    User Values are:
    0 = Not Used, 1 = FIC-21-1, 2 = EV-2, 3 = EV-3, 4 = AG-4, 5 = FIC-21-2, 6 = FIC-21-3, 7 = FIC-21-4, 8 = FIC-46-1, 9 = EV-42, 10 = EV-20
  N24:12: This Rung Calculates
    the Range Values for PID Statements, Analog Inputs and Analog Outputs
    These are used Elsewhere in PLC Logic to calulate either
    other Units
    (PID Statement Inputs, Analog Output Values, etc)
  N24:20: This Rung Calculates the PLC Ranges as Shown
    For use elsewhere in the PLC Program
  N50:0/0: This Rung Stops EV-1 Rotor Drive
    when the operator presses the EV-1 PB
    AND the motor is Off
    OR
    The Interlocks are NOT satisfied
  N50:2/0: This Rung determines the status of the Interlocks for EV-1 Rotor Drive
  N50:4/0: This rung sets a 1-shot bit whenever EV-1 Rotor Drive
    is Started
  N50:5/13: This rung sets a 1-shot bit whenever EH-24 Hot Oil Heater
    HMI Start/Stop PB
    is Pressed
  N50:6/0: This rung sets a 1-shot bit whenever EV-1 Rotor Drive
    is Stopped
  N50:15/11: This Rung Resets All
    HMI PB's to
    0 State to allow their next use to be detected
    (This is required due to iFIX's inability to generate momentary PB's, not required for PanelView Plus)
  N50:16/11: This Rung Generates a 1-shot
    whenever the Operator
    presses the FIC-21-1 Output Select PB
  N50:20: This rung resets any
    iFIX Momentary PB's to 0
    (ifix does not have momentary PB Feature)
  N50:41/14: This rung sets a 1-shot bit whenever
    the EV-2 Residue
    Calculate Flow Rate PB
    is Pressed
  N61:0/[N23:82]: This Rung Starts EV-2 Rotor Drive
    when the operator presses the EV-2 PB
    AND
    the Interlocks are satisfied and the motor is Off
  N101:20/0: DELETE THIS RUN FOR REAL PLC
  N213:1: This Rung Converts the Output from
    PIC-28-1
    Steam Pressure Controller
    to Open PV-28-1 (Steam Valve) Between 0% to 100% .
    PV-28-1 Fails Closed
  N213:3: This Rung Split Ranges the Output from
    TIC-11-1
    Tempered Water Loop No-1
    to Close TV-11-1 (Cooling Valve) Between 0% to 50% while keeping TV-11-2 (Heating Valve) Closed.
    then
    to Open TV-11-2 (Heating Valve) Between 50% to 100% while keeping TV-11-1 (Cooling valve) Closed.
    At  50%, Both Valves are Closed
      TV-11-1 Fails Open, TV-11-2 Fails Closed
  N214:0: This Rung Converts the Output from
    TIC-12-1
    Tempered Water Loop No-2
    to Close TV-12-1 (Cooling Valve) Between 0% to 100% .
    TV-12-1 Fails Open
  N214:1: This Rung Converts the Output from
    TIC-15-1
    Tempered Oil Loop No-1
    to Open TV-15-1 (Heating Valve) Between 0% to 100% .
    TV-15-1 Fails Closed
  N214:3: This Rung Converts the Output from
    TIC-24-1
    Hot Oil Loop
    to Increase the Firing Rate of TY-24-1 (Heater SCR Controller) Between 0% to 100% .
    TY-24-1 is Off 100% at 0%, On 50% of time at 50% and On 100% of time at 100%.
  N215:0: This Rung Sends the
    EV-2 Rotor Speed Setpoint
    to the VFD which controls its speed.
    A 1-shot is used when the motor is started to set an initial speed
    A 1-shot is also used when it is stopped to reset the speed to 0.0
    and the last rung actually passed the speed signal to the analog output module which sontrols the motors speed
  N215:1: This Rung Sends the
    EV-3 Rotor Speed Setpoint
    to the VFD which controls its speed.
    A 1-shot is used when the motor is started to set an initial speed
    A 1-shot is also used when it is stopped to reset the speed to 0.0
    and the last rung actually passed the speed signal to the analog output module which sontrols the motors speed
  N215:2: This Rung Sends the
    AG-4 Agitator Speed Setpoint
    to the VFD which controls its speed.
    A 1-shot is used when the motor is started to set an initial speed
    A 1-shot is also used when it is stopped to reset the speed to 0.0
    and the last rung actually passed the speed signal to the analog output module which sontrols the motors speed
  N216:1: This Rung Moves the
    FIC-21-1 PID Output to the
    Selected Pump VFD Speed Control Based on which Pump is Connected to the Feed Flow Loop
  N216:3: This Rung Moves the
    PIC-30-1 PID Output to Pump PU-30's VFD Speed Control
  N218:0: This Rung Copies Setup Data for all TE's
    to their Output Addresses when the PLC is first placed in the Run Mode
    This Information determines that the TE data returned from the Input modules will
    use °C Units for a Type "J" Thermocouple
  O:6.16/0: This Rung Starts PU-13 Tempered Oil Pump No-2
    when the operator presses the PU-13 PB
    AND
    the Interlocks are satisfied and the motor is Off
  O:6.19/4: This Rung Starts PU-13 Tempered Oil Pump No-2
    when the operator presses the PU-13 PB
    AND
    the Interlocks are satisfied and the motor is Off
  O:15.0: This Rung Controls the Status and Speed of
    VFD02
    if it's controls are enabled
  O:15.1: This Rung Controls the Status and Speed of
    VFD03
    if it's controls are enabled
  O:15.2: This Rung Controls the Status and Speed of
    VFD04
    if it's controls are enabled
  O:15.3: This Rung Controls the Status and Speed of
    VFD01
    if it's controls are enabled
  O:23.0/0: This Rung Stops EV-1 Rotor Drive
    when the operator presses the EV-1 PB
    AND the motor is Off
    OR
    The Interlocks are NOT satisfied
  O:23.0/11: This Rung Starts PU-23 Hot Oil Pump
    when the operator presses the PU-23 PB
    AND
    the Interlocks are satisfied and the motor is Off
  O:23.0/12: This Rung Starts EH-24 Hot Oil Heater
    when the operator presses the EH-24 PB
    AND the Heater is Off
    AND
    The Interlocks are satisfied
  Q62:1: This Rung Enables EH-24, Hot Oil Heater
    when the operator presses the EH-24 PB
    AND
    the Interlocks are satisfied and the Contatcer is Off
     (The Jump Stattement is required since this device does Not have a feedback connection from contactor to indicate actual status,
    because of this, an internal bit is used.  When an internal bit is used, the next statement (Stop/disable)
    will immediantely be executed, resulting in the motor/contactor not being de-energized.  The Jump statement eliminates this problem)
  Q64:1: This Rung Enables EH-27, Hot Oil SuperHeater
    when the operator presses the EH-27 PB
    AND
    the Interlocks are satisfied and EH-27 is disabled
      (The Jump Stattement is required since this device does Not have a feedback connection from contactor to indicate actual status,
    because of this, an internal bit is used.  When an internal bit is used, the next statement (Stop/disable)
    will immediantely be executed, resulting in the motor/contactor not being de-energized.  The Jump statement eliminates this problem)
  T4:31: This Rung Sets a bit when
    PT-26-1 is less than PSL-26-1's Setpoint.
    Used to enable VB-26
  T51:0: This run starts a timer whenever EV-1 Rotor Drive
    is started to verify that it actually starts within 5 sec's
    If Not, then it is assumed that the motor's O.l.s have tripped
  T51:1: This run starts a timer whenever EV-2 Rotor Drive
    is started to verify that it actually starts within 5 sec's
    If Not, then it is assumed that the motor's O.l.s have tripped
  T51:2: This run starts a timer whenever EV-3 Rotor Drive
    is started to verify that it actually starts within 5 sec's
    If Not, then it is assumed that the motor's O.l.s have tripped
  T51:3: This run starts a timer whenever AG-4 Feed Tank Agitator
    is started to verify that it actually starts within 5 sec's
    If Not, then it is assumed that the motor's O.l.s have tripped
  T51:4: This run starts a timer whenever VP-9 Beach-Ross Vacuum Pump
    is started to verify that it actually starts within 5 sec's
    If Not, then it is assumed that the motor's O.l.s have tripped
  T51:5: This run starts a timer whenever VP-10 Kinney Vacuum Pump
    is started to verify that it actually starts within 5 sec's
    If Not, then it is assumed that the motor's O.l.s have tripped
  T51:6: This run starts a timer whenever PU-11 Tempered Water Pump No-1
    is started to verify that it actually starts within 5 sec's
    If Not, then it is assumed that the motor's O.l.s have tripped
  T51:7: This run starts a timer whenever PU-12 Tempered Water Pump No-2
    is started to verify that it actually starts within 5 sec's
    If Not, then it is assumed that the motor's O.l.s have tripped
  T51:8: This run starts a timer whenever PU-15 Tempered Oil Pump
    is started to verify that it actually starts within 5 sec's
    If Not, then it is assumed that the motor's O.l.s have tripped
  T51:9: This run starts a timer whenever PU-21 Feed Pump No-1
    is started to verify that it actually starts within 5 sec's
    If Not, then it is assumed that the motor's O.l.s have tripped
  T51:10: This run starts a timer whenever PU-22 Feed Pump No-2
    is started to verify that it actually starts within 5 sec's
    If Not, then it is assumed that the motor's O.l.s have tripped
  T51:11: This run starts a timer whenever PU-23 Hot Oil Pump
    is started to verify that it actually starts within 5 sec's
    If Not, then it is assumed that the motor's O.l.s have tripped
  T51:13: This run starts a timer whenever VB-26 Roots Vacuum Blower
    is started to verify that it actually starts within 5 sec's
    If Not, then it is assumed that the motor's O.l.s have tripped
  T51:15: This run starts a timer whenever PU-30 City Water Booster Pump
    is started to verify that it actually starts within 5 sec's
    If Not, then it is assumed that the motor's O.l.s have tripped
  T51:16: This run starts a timer whenever  VB-35 TutHill Vacuum Blower
    is started to verify that it actually starts within 5 sec's
    If Not, then it is assumed that the motor's O.l.s have tripped
  U:3: This Rung Calls the Subroutine Files Listed
  U:10: This Rung Calls the Subroutine Files Listed
  U:31: This Rung Calls the Subroutine Files Listed
  U:59: This Rung Calls the Subroutine Files Listed
  U:66: This Rung Calls the Subroutine Files Listed
  U:101: DELETE THIS RUNG AND FILE WHEN USING THE REAL PLC CONFIGURATION WITH REAL I/O

REVISION NOTES
  0: Totalizer Updates for Harting Test

DATA TABLE (non-zero values as saved)
DATA B3
% B3:0 % 0X007E 0X0000 0X0000 0X0000 0X0000 0X000C 0X0000 0X0000 0X0000 0X0000
% B3:10 % 0X9000 0X0000 0X0002 0X0000 0X0000 0X0000 0X0000 0X0000 0X0000 0X0000
% B3:20 % 0X0000 0X0000 0X0002 0X0000 0X0000 0X0000 0X0000 0X0000 0X0000 0X0000
% B3:30 % 0X0009 0X0000 0X0000 0X0000 0X0009 0X0000 0X0000 0X0000 0X0000 0X0000
% B3:70 % 0X0028 0X0000 0X0000 0X0000 0X0000 0X0000 0X0000 0X0000 0X0000 0X0000
DATA T4
% .PRE .ACC %
% T4:0 % 150 0
% T4:1 % 3000 1418
% T4:2 % 3600 1529
% T4:3 % 1000 0
% T4:4 % 100 0
% T4:6 % 1 0
% T4:11 % 6000 0
% T4:12 % 6000 0
% T4:13 % 6000 0
% T4:14 % 6000 0
% T4:21 % 10 10
% T4:22 % 50 30
% T4:23 % 10 10
% T4:24 % 50 30
% T4:25 % 30 30
% T4:26 % 12 6
% T4:30 % 5 0
% T4:31 % 5 5
% T4:32 % 2 0
% T4:34 % 5 0
% T4:35 % 1 0
DATA C5
% .PRE .ACC %
% C5:0 % 3600 1446
% C5:1 % 16000 -19876
% C5:2 % 16000 0
% C5:3 % 16000 21413
% C5:4 % 16000 21419
% C5:5 % 16000 21249
% C5:6 % 16000 21298
% C5:7 % 16000 2
% C5:8 % 16000 22936
% C5:11 % 600 0
% C5:12 % 600 0
% C5:13 % 600 600
% C5:14 % 600 0
DATA N7
% N7:0 % 4 7 2014 0 0 0 0 0 0 0
DATA F8
% F8:0 % 100 200 0 0 0
DATA N11
% N11:0 % 0 277 253 259 300 7599 7599 7599 7599 7599
% N11:10 % 267 274 275 298 282 7599 7599 7599 7599 315
% N11:20 % 315 263 264 265 256 275 7599 264 265 170
% N11:30 % 187 204 259 286 283 282 284 0 0 0
% N11:100 % 6 15152 0 16383 16383 12197 0 0 0 16383
% N11:120 % 1500 50 1950 600 50 10000 750 0 10000 10000
% N11:130 % 0 13313 8018 1564 0 0 0 0 0 0
% N11:150 % 0 2000 1000 1500 0 0 0 0 0 0
% N11:190 % 0 1000 0 0 0 0 0 0 0 0
% N11:220 % 0 5000 6000 5000 6000 6000 6000 0 0 0
DATA N12
% N12:0 % 0 170 187 204 259 286 283 282 284 0
% N12:10 % 128 0 0 0 0 0 0 0 0 0
% N12:20 % 0 0 8 8 8 8 8 8 0 0
% N12:100 % 0 0 0 0 0 0 0 0 -32768 0
% N12:110 % 0 0 0 0 0 0 0 0 -32768 0
% N12:120 % 15 0 0 0 0 0 0 0 0 0
DATA N13
% N13:0 % 0 3136 3136 3136 3136 3136 3136 3136 3136 3136
% N13:10 % 3136 3136 3136 3136 3136 3136 3136 3136 3136 3136
% N13:20 % 3136 3136 3136 3136 3136 3136 3136 3136 3136 0
% N13:30 % 0 13107 13107 0 0 0 0 0 0 0
% N13:40 % 255 0 0 0 0 0 0 0 0 0
% N13:50 % 0 0 0 0 15 3840 0 0 0 0
% N13:70 % 0 0 0 0 15 3840 0 0 0 0
% N13:100 % -256 0 0 0 0 0 0 0 0 0
% N13:110 % -256 0 0 0 0 0 0 0 0 0
% N13:120 % 0 0 0 0 15 3840 0 0 0 0
DATA F14
% F14:5 % 40 30 0 0 0
% F14:10 % 45 0 0 0 0
DATA N15
% N15:0 % -24566 0 0 8 5 10 0 6000 0 0
% N15:10 % 0 60 0 15 0 0 0 0 -5805 0
% N15:20 % 0 0 0 0 0 40 1 0 5000 7500
% N15:30 % -24574 0 0 7 5 11 0 6000 0 0
% N15:40 % 0 60 0 15 0 0 0 0 7241 0
% N15:60 % -24570 0 0 50 3 0 0 1950 0 0
% N15:70 % 0 100 0 15 0 0 100 16383 0 0
% N15:80 % 0 0 0 0 0 0 0 2500 5000 7500
% N15:90 % -24570 0 7444 100 10 0 0 10000 0 0
% N15:100 % 0 100 0 15 7444 0 80 13086 29382 2
% N15:110 % -1456 0 7444 0 12197 0 0 0 0 0
% N15:150 % -24318 0 1580 2 5 0 0 2000 0 10
% N15:160 % 0 100 0 15 1580 2 50 8192 -12210 3
% N15:170 % 10592 0 1582 0 13313 0 0 500 1000 1500
% N15:180 % -24566 0 377 20 10 0 0 1000 0 0
% N15:190 % 0 83 0 15 377 5 0 -156 -28170 1
% N15:200 % -31472 0 381 0 8018 0 0 250 500 750
DATA N16
% N16:0 % -24566 0 0 8 5 10 0 6000 0 0
% N16:10 % 0 60 0 15 0 0 0 0 -24274 0
% N16:20 % 0 0 0 0 0 0 0 950 1900 2850
% N16:30 % -24314 0 0 10 5 0 0 5000 0 0
% N16:40 % 0 60 0 15 0 0 0 0 -2178 0
% N16:50 % 0 0 0 0 0 0 0 1500 3000 4500
% N16:60 % -24318 0 143 100 5 0 0 1500 0 0
% N16:70 % 0 60 0 15 143 0 0 0 9388 0
% N16:80 % 25024 0 143 0 1564 0 0 750 1500 2250
% N16:150 % -24570 0 0 100 3 0 0 1000 0 0
% N16:160 % 0 60 0 15 0 0 0 0 0 0
DATA N17
% N17:0 % -24318 0 170 15 3 0 11468 2000 0 0
% N17:10 % 0 100 0 15 170 0 50 -3276 30726 0
% N17:20 % 22288 0 170 0 1393 50 0 0 0 0
% N17:30 % -24318 0 259 20 3 0 0 2000 0 0
% N17:40 % 0 100 0 15 259 0 50 8192 25776 0
% N17:50 % -31584 0 259 0 2122 50 0 0 0 0
% N17:60 % -24318 0 286 250 20 5 0 3500 0 0
% N17:70 % 0 100 0 15 286 0 0 40 20578 0
% N17:80 % 21485 0 286 0 1325 0 0 0 0 0
% N17:90 % -24566 0 283 900 400 0 0 3500 0 0
% N17:100 % 0 100 0 15 283 0 0 450 -2237 0
% N17:110 % 21264 0 283 0 1329 0 3430 0 0 0
% N17:120 % -24574 0 280 30 30 0 0 3500 0 0
% N17:130 % 0 100 0 15 280 0 0 3 1632 0
% N17:140 % 20976 0 280 0 1320 0 0 0 0 0
% N17:150 % -24318 0 264 100 30 5 0 3500 0 0
% N17:160 % 0 100 0 15 264 0 0 0 -10202 0
% N17:170 % 19776 0 264 0 1236 0 0 0 0 0
DATA N18
% N18:0 % 0 0 0 0 0 16383 13106 0 8192 0
% N18:10 % 0 0 16383 16383 0 0 0 0 0 0
% N18:20 % 0 8192 8192 0 0 0 0 0 0 0
DATA N20
% N20:0 % 0 51 51 0 0 0 0 0 0 0
% N20:30 % -5 -5 -5 -5 -5 -5 -5 -5 0 0
DATA F21
% F21:0 % 0 27.7 25.3 25.9 30
% F21:5 % 759.9 759.9 759.9 759.9 759.9
% F21:10 % 26.7 27.4 27.5 29.8 28.2
% F21:15 % 759.9 759.9 759.9 759.9 31.5
% F21:20 % 31.5 26.3 26.4 26.5 25.6
% F21:25 % 27.5 759.9 26.4 26.5 17
% F21:30 % 18.7 20.4 25.9 28.6 28.3
% F21:35 % 28.2 28.4 0 0 0
% F21:50 % 0 162.521 48.93941 14.31787 0
% F21:60 % 0 -0.1526019 5.859911 -0.2289028 0
% F21:65 % 0 0 0.01526019 -50.02289 -15.00229
% F21:70 % 0.3815047 4.624218 -48.74256 61.95483 5.156798
% F21:75 % 744.4682 77.43781 0 -0.3571429 1258.202
% F21:80 % -250.0381 3604.48 2621.44 0.025 0
% F21:95 % 0 0 83417.15 0.0038 205.7111
% F21:120 % 0 0.01159703 0.01373333 -0.0006103702 0.002746666
% F21:125 % 0 0.003204639 0 0 0.001495453
% F21:130 % 0 -0.07630093 -0.04578056 -0.1144514 -9.385015
% F21:135 % 0 -2.563711 0 0 0
% F21:140 % 0 0.2499619 0.4996948 0.4938959 0.4841294
% F21:145 % 0.4997711 0.4937433 0 0 0
% F21:160 % 29.75736 0 0 0 0
% F21:170 % 0 0 0 0.002929777 0.003906369
% F21:175 % 0 0 0 0.001953185 0
% F21:180 % 0.007202368 0 0 0 0
% F21:195 % 0 0 0 0 199.76
% F21:200 % 0 -25.00381 0 0 0
% F21:205 % 0 -50.00763 0 0 0
DATA F22
% F22:0 % 22.22 27.45 0 0 0
% F22:10 % 0 4.624218 0.3815047 61.95483 0
% F22:20 % 0 0.3815047 0.3815047 0.3815047 0
% F22:50 % 0 26.7 26.4 26.5 26.3
% F22:55 % 0 26.7 27.5 27.7 0
% F22:60 % 0 28.2 759.9 759.9 27.4
% F22:65 % 26.7 25.6 31.5 26.5 0
% F22:70 % 0 26.3 26.7 26.5 25.6
% F22:75 % 27.5 759.9 26.4 26.5 0
% F22:90 % 0 26.7 25.9 28.6 28.3
% F22:95 % 28.2 28.4 0 0 0
% F22:100 % 0 759.9 759.9 25.9 27.5
% F22:110 % 0 25.3 27.7 0 0
% F22:120 % 0 17 0 0 0
% F22:130 % 0 25.9 0 0 0
% F22:140 % 0 28.3 28.2 26.4 0
% F22:180 % 0 28.4 0 0 0
% F22:190 % 0 759.9 31.5 0 0
% F22:200 % 26.4 26.4 26.4 26.4 27.5
% F22:205 % 0 27.5 31.5 0 0
% F22:210 % 0 -0.04578056 -0.07630093 0 0
% F22:220 % 0 -0.1144514 0 -0.07630093 0
% F22:230 % 0 -0.1144514 -0.1144514 -0.1144514 0
DATA N23
% N23:0 % 0 24 6 10 36 1 0 0 0 0
% N23:10 % 0 2 5 0 0 0 0 0 0 0
% N23:20 % 0 2 5 6 3 0 0 0 0 0
% N23:30 % 0 2 1 0 3 0 1 3 3 3
% N23:40 % 7 132 131 130 133 130 131 133 133 133
% N23:50 % 0 1 0 3 0 0 0 0 0 0
% N23:60 % 11 71 70 73 70 70 70 0 0 0
% N23:70 % 8 0 0 1 0 8 0 0 0 0
% N23:80 % 9 0 2 3 4 0 5 0 0 0
% N23:90 % 0 6 2 3 4 10 0 0 8 0
% N23:100 % 0 10 27 23 21 0 10 25 1 14
% N23:110 % 15 16 11 10 24 19 23 21 10 23
% N23:120 % 24 25 26 27 28 0 0 0 10 32
% N23:130 % 33 34 5 6 3 25 2 1 0 0
% N23:140 % 29 3 34 0 0 0 0 0 0 0
% N23:150 % 0 0 36 17 20 0 0 35 36 0
% N23:160 % 12 19 0 0 0 0 0 0 0 0
% N23:170 % 35 27 27 27 27 27 25 0 0 0
% N23:210 % 0 130 130 130 130 130 130 0 0 0
% N23:220 % 2 1 0 0 0 0 0 0 0 0
% N23:240 % 0 1 1 1 1 0 0 0 0 0
% N23:250 % 0 4 0 0 0 0
DATA N24
% N24:0 % 3277 16383 13106 0 0 0 32767 32767 0 0
% N24:10 % 6240 31400 25160 0 30850 30850 0 0 0 0
% N24:20 % 0 16383 16383 8192 0 0 0 0 0 0
% N24:30 % 7000 19000 0 0 0 0 0 0 0 0
% N24:40 % 11 30600 30800 0 0 0 0 0 0 0
% N24:50 % 0 0 0 0 0 31 31 255 63 0
DATA N25
% N25:0 % 0 3 0 0 0 -24448 11 0 0 0
% N25:10 % -15322 1 9 0 0 -15194 9 9 0 0
% N25:20 % -23512 14 14 0 0 9384 1 14 0 0
% N25:30 % -23510 14 14 0 0 9386 1 14 0 0
% N25:50 % 11 8 0 0 0 0 0 0 0 0
% N25:80 % 3 0 4 0 0 0 0 0 0 0
% N25:90 % 1 1 3 0 0 0 0 0 0 0
% N25:100 % 1026 1 9 0 0 9346 9 9 0 0
% N25:110 % 1028 1 9 0 0 9348 9 9 0 0
% N25:120 % -24570 14 0 0 0 8326 1 0 0 0
DATA F26
% F26:0 % 32768 -32768 0 0 0
% F26:5 % -25 350.5 0 0 0
% F26:10 % 0 5 5 1.25 2.5
% F26:15 % 3.75 0 0 0 0
% F26:20 % 0 195 195 48.75 97.5
% F26:25 % 146.25 0 0 0 0
% F26:30 % 0 60 60 15 30
% F26:35 % 45 0 0 0 0
% F26:40 % 0 5 5 1.25 2.5
% F26:45 % 3.75 0 0 0 0
% F26:50 % 0 1000 1000 250 500
% F26:55 % 750 0 0 0 0
% F26:60 % 0 75 75 18.75 37.5
% F26:65 % 56.25 0 0 0 0
% F26:70 % 0 1000 1000 250 500
% F26:75 % 750 0 0 0 0
% F26:80 % 0 1000 1000 250 500
% F26:85 % 750 0 0 0 0
% F26:90 % 0 1000 1000 250 500
% F26:95 % 750 0 0 0 0
% F26:100 % 0 150 150 37.5 75
% F26:105 % 112.5 0 0 0 0
% F26:110 % 0 500 500 125 250
% F26:115 % 375 0 0 0 0
% F26:120 % 0 600 600 150 300
% F26:125 % 450 0 0 0 0
% F26:130 % 0 500 500 125 250
% F26:135 % 375 0 0 0 0
% F26:140 % 0 600 600 150 300
% F26:145 % 450 0 0 0 0
% F26:150 % 0 600 600 150 300
% F26:155 % 450 0 0 0 0
% F26:160 % 0 200 200 50 100
% F26:165 % 150 0 0 0 0
% F26:170 % 0 100 100 25 50
% F26:175 % 75 0 0 0 0
% F26:180 % 0 600 600 150 300
% F26:185 % 450 0 0 0 0
% F26:190 % 0 200 200 50 100
% F26:195 % 150 0 0 0 0
% F26:200 % 0.5 1.5 1 0.75 1
% F26:205 % 1.25 0 0 0 0
% F26:210 % 0 150 150 37.5 75
% F26:215 % 112.5 0 0 0 0
% F26:220 % 0 200 200 50 100
% F26:225 % 150 0 0 0 0
% F26:230 % 0.5 1.5 1 0.75 1
% F26:235 % 1.25 0 0 0 0
% F26:240 % 0.5 1.5 1 0.75 1
% F26:245 % 1.25 0 0 0 0
DATA F27
% F27:0 % 360448 262144 0 0 0
% F27:10 % 6.250191 15151.71 -4095.125 16916.77 16896.77
% F27:15 % 12196.62 -70.00214 0 -5.851071 20613.13
% F27:20 % 0 -2.500076 -1.250038 -3.750114 -256.2578
% F27:25 % 0 -70.00214 0 0 0
% F27:30 % 1392.555 2121.599 1324.683 1329.363 1320.002
% F27:35 % 1235.746 0 0 0 0
% F27:40 % 0 13312.91 8017.745 1563.798 0
% F27:45 % 25 35 0 0 0
% F27:50 % 0 30 50 0 0
% F27:60 % 0 150 200 50 4
% F27:65 % 4 4 30 30 0
% F27:70 % 0 55 45 250 120
% F27:75 % 311 250 0 0 25
% F27:80 % 0 297 297 20 2
% F27:90 % 0 -4096.375 0 0 0
% F27:100 % 0 0 -28.25 0.018 1471.6
% F27:105 % 0 3604.48 2649.69 0.007000001 -1471.6
% F27:110 % 22 2293.76 -141.65 -0.013 -49.4
% F27:115 % 66 2293.76 -182.2 0.025 -49.5
% F27:120 % 60 0.02066667 0.02916667 600 0.02916667
% F27:125 % 44 0 83417.15 0.0038 205.7111
% F27:130 % 0 124 175 0 175
% F27:140 % 0 0 0 3.813 3.818
% F27:145 % 0 0 0 6.534 18.795
% F27:150 % 0 0 0 5 5
% F27:155 % 0 0.0001 0.0001 0.0001 0.0001
% F27:160 % 0 0.0001 0.0001 300.0001 300.0001
% F27:165 % 0 0 0 32.65199 179.7239
% F27:180 % 0 10 0 0 0
% F27:200 % 0 0 0 0 0.05555556
% F27:205 % 0 0 82.00242 0 0
DATA F28
% F28:0 % 0 3604.48 2621.44 0.025 0
DATA F29
% F29:0 % 0 150 300 450 600
% F29:5 % 0 0 600 0 0
% F29:10 % 0 150 300 450 600
% F29:15 % 0 0 600 0 0
% F29:20 % 0 150 300 450 600
% F29:25 % 0 0 600 0 0
% F29:30 % 0 125 250 375 500
% F29:35 % 0 0 500 0 0
% F29:40 % 0 37.5 75 112.5 1500
% F29:45 % 14.3 0 150 0 14.3
% F29:50 % 0 48.75 97.5 146.25 195
% F29:55 % 0 0 195 100 0
% F29:60 % 0 250 500 750 1000
% F29:65 % 744.4 0 1000 80 744.4
% F29:70 % 0 50 100 150 200
% F29:75 % 158 0 200 50 158
% F29:80 % 0 25 50 75 100
% F29:85 % 37.7 0 100 0 37.7
% F29:90 % 0 900 1800 2700 3600
% F29:95 % 0 0 3600 0 0
% F29:100 % 0 74.25 148.5 222.75 297
% F29:105 % 0 60 297 0 0
% F29:110 % 0 135 270 405 540
% F29:115 % 0 60 540 0 0
% F29:120 % 0 29.25 58.5 87.75 117
% F29:125 % 0 60 117 0 0
% F29:130 % 0 15 30 45 60
% F29:135 % 0 60 60 0 0
% F29:140 % 0 15 30 45 60
% F29:145 % 0 60 60 0 0
% F29:150 % 0 50 100 150 200
% F29:155 % 17 0 200 50 17
% F29:160 % 0 50 100 150 200
% F29:165 % 25.9 0 200 50 25.9
% F29:170 % 0 87.5 175 262.5 350
% F29:175 % 28.6 0 350 0 28.6
% F29:180 % 0 87.5 175 262.5 350
% F29:185 % 28.3 0 350 0 28.3
% F29:190 % 0 87.5 175 262.5 350
% F29:195 % 28 0 350 0 28
% F29:200 % 0 87.5 175 262.5 350
% F29:205 % 26.4 0 350 0 26.4
% F29:210 % 0 15 30 45 60
% F29:215 % 0 60 60 0 0
% F29:220 % 0 25 50 75 100
% F29:225 % 0 0 100 0 0
DATA F30
% F30:0 % 0 10 10 2.5 5
% F30:5 % 7.5 0 0 0 0
% F30:10 % 0.5 1.5 1 0.75 1
% F30:15 % 1.25 0 0 0 0
% F30:20 % 0.5 1.5 1 0.75 1
% F30:25 % 1.25 0 0 0 0
% F30:30 % 0.5 1.5 1 0.75 1
% F30:35 % 1.25 0 0 0 0
% F30:40 % 0 0.875 1.75 2.625 3.5
% F30:45 % 5.25 0 3.5 0 0
% F30:50 % 0 15 30 45 60
% F30:55 % 0 60 60 0 0
% F30:60 % 0 15 30 45 60
% F30:65 % 0 60 60 0 0
% F30:70 % 0 15 30 45 60
% F30:75 % 0 60 60 0 0
% F30:80 % 0 74.25 148.5 222.75 297
% F30:85 % 0 60 297 0 0
% F30:90 % 0 74.25 148.5 222.75 297
% F30:95 % 0 60 297 0 0
% F30:110 % 0 2.75 5.5 8.25 11
% F30:115 % 0 0 11 0 0
% F30:120 % 0 4 8 12 16
% F30:125 % 0 0 16 0 0
% F30:130 % 0 3 6 9 12
% F30:135 % 0 0 12 0 0
% F30:140 % 0 4 8 12 16
% F30:145 % 0 0 16 0 0
% F30:150 % 0 2 4 6 8
% F30:155 % 0 0 8 0 0
% F30:160 % 0 1.775 3.55 5.325 7.1
% F30:165 % 0 0 7.1 0 0
% F30:170 % 0 2 4 6 8
% F30:175 % 0 0 8 0 0
% F30:180 % 0 7.375 14.75 22.125 29.5
% F30:185 % 0 0 29.5 0 0
% F30:200 % 5 1 3 0.75 1
% F30:205 % 0 0 2 5 10
% F30:210 % 0.75 0 0 0 0
% F30:220 % 0 25 50 75 100
% F30:225 % 0 0 100 0 0
% F30:230 % 0 50 100 150 200
% F30:235 % 0 0 200 0 0
DATA N50
% N50:0 % 0 0 -30209 974 0 0 0 0 0 256
% N50:10 % -1 1791 0 0 0 0 0 0 0 0
DATA T51
% .PRE .ACC %
% T51:0 % 5 0
% T51:1 % 5 0
% T51:2 % 600 0
% T51:3 % 5 0
% T51:4 % 5 0
% T51:5 % 5 0
% T51:6 % 5 0
% T51:7 % 5 0
% T51:8 % 5 0
% T51:9 % 5 0
% T51:10 % 5 0
% T51:11 % 5 0
% T51:13 % 5 0
% T51:14 % 20 0
% T51:15 % 5 0
% T51:16 % 5 0
% T51:17 % 10 0
% T51:18 % 5 0
% T51:19 % 5 0
% T51:20 % 5 0
% T51:21 % 60 0
% T51:22 % 60 0
% T51:23 % 60 0
% T51:24 % 60 0
% T51:25 % 60 0
% T51:26 % 60 0
% T51:27 % 60 0
% T51:28 % 60 0
% T51:29 % 500 500
% T51:30 % 5 0
% T51:31 % 5 0
% T51:33 % 5 0
% T51:34 % 5 0
% T51:37 % 5 0
% T51:38 % 5 0
% T51:41 % 1200 0
% T51:50 % 200 0
% T51:58 % 200 0
% T51:59 % 200 0
% T51:60 % 200 0
% T51:70 % 20 0
% T51:71 % 20 0
% T51:72 % 20 0
% T51:73 % 20 0
% T51:81 % 5 0
DATA F52
% F52:0 % 2 1.5 1 2 1.5
% F52:5 % 1 0 0 0 0
% F52:10 % 140 150 140 150 0
DATA F62
% F62:0 % 0 0 0 0.002929777 0.003906369
% F62:5 % 0.001953185 0.001733451 0.001953185 0.007202368 0
DATA F63
% F63:0 % 0 3 10 7.5 10
% F63:5 % 5 2 5 10 0
DATA N100
% N100:0 % 16 0 0 0 0 0 0 0 0 0
DATA N101
% N101:0 % 0 0 108 -11261 108 -11262 0 0 0 0
% N101:10 % 0 0 0 0 18236 9397 29241 19589 209 25080
% N101:20 % 146 28320 0 0 0 0 0 0 0 0
% N101:40 % 0 0 0 0 2 0 -17204 11472 2610 8306
% N101:50 % 7 7 0 48 30 0 0 0 0 0
DATA F201
% F201:0 % 0 -0.07630093 -0.07630093 -0.07630093 -0.07630093
% F201:5 % -0.07630093 -0.07630093 -0.07630093 -0.07630093 -0.07630093
% F201:10 % -0.07630093 0 0 0 0
% F201:50 % -0.07630093
DATA F202
% F202:0 % 0 -0.04578056 -0.04578056 -0.04578056 -0.04578056
% F202:5 % -0.04578056 -0.04578056 -0.04578056 -0.04578056 -0.04578056
% F202:10 % -0.04578056 0 0 0 0
% F202:50 % -0.04578056
DATA F203
% F203:0 % 0 -0.1144514 -0.1144514 -0.1144514 -0.1144514
% F203:5 % -0.1144514 -0.1144514 -0.1144514 -0.1144514 -0.1144514
% F203:10 % -0.1144514 0 0 0 0
% F203:50 % -0.1144514
DATA F204
% F204:0 % 0 -9.385015 -9.385015 -9.385015 -9.385015
% F204:5 % -9.385015 -9.385015 -9.385015 -9.385015 -9.385015
% F204:10 % -9.385015 0 0 0 0
% F204:50 % -9.385015
DATA F206
% F206:0 % 0 -2.563711 -2.563711 -2.563711 -2.563711
% F206:5 % -2.563711 -2.563711 -2.563711 -2.563711 -2.563711
% F206:10 % -2.563711 0 0 0 0
% F206:50 % -2.563711
